FUNCTION_BLOCK WaterTank
  (* Standard: 61499-2 *)
  (* Version 0.1, 2015-00-10, syy, syy-PC *)
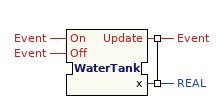
  EVENT_INPUT
    On;
    Off;
  END_EVENT
  EVENT_OUTPUT
    Update WITH x;
  END_EVENT
  VAR_OUTPUT
    x : REAL;
  END_VAR
  VAR
    C1x : REAL;
    k : REAL;
    d : REAL;
  END_VAR
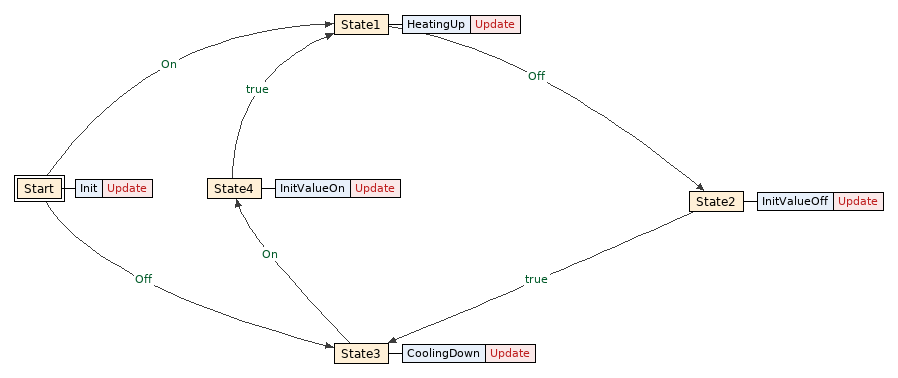
  EC_STATES
    Start : Init -> Update;
    State1 : HeatingUp -> Update;
    State2 : InitValueOff -> Update;
    State3 : CoolingDown -> Update;
    State4 : InitValueOn -> Update;
  END_STATES
  EC_TRANSITIONS
    Start TO State1 := On;
    Start TO State3 := Off;
    State1 TO State2 := Off;
    State2 TO State3 := true;
    State3 TO State4 := On;
    State4 TO State1 := true;
  END_TRANSITIONS
  ALGORITHM Init IN C:
me->x = 20;
me->C1x = -130;
me->d = 0.01;
me->k = 1;
  END_ALGORITHM
  ALGORITHM HeatingUp IN C:
//me->x = (float) me->C1x*exp(-0.075*me->d*me->k) + 150.0;
me->x = 100;
me->k++;
printf("Temperature : %f\n", me->x);
  END_ALGORITHM
  ALGORITHM InitValueOff IN C:
me->k=0;
me->C1x=me->x;
  END_ALGORITHM
  ALGORITHM CoolingDown IN C:
//me->x = (float) me->C1x*exp(-0.075*me->d*me->k);
me->x = 20;
me->k++;
printf("Temperature : %f\n", me->x);
  END_ALGORITHM
  ALGORITHM InitValueOn IN C:
me->k=0;
me->C1x=me->x-150;
  END_ALGORITHM
END_FUNCTION_BLOCK
